{attribute 'GeneratedUsingTerminal: EK1100-0000-0018'}
{attribute addProperty BoxType "EK1100-0000-0018"}
{attribute addProperty Id "Beckhoff_EL72xxEK1122Beckhoff_EL72xxEK1122_A6E7F55E2A_0001_EL7201_0000_0017EL7201_91DE43F025A_0002_EL7201_0000_0018EL7201_91DE43F025A_0003_EL7201_0000_0019EL7201_91DE43F025A_0004_EL7201_0000_0020EL7201_91DE43F025A_0005_EL7201_0000_0021EL7201_91DE43F025A_0006_EL7201_0001_0017EL7201_24495B2825A_0007_EL7201_0001_0018EL7201_24495B2825A_0008_EL7201_0001_0019EL7201_24495B2825A_0009_EL7201_0001_0020EL7201_24495B2825A_0010_EL7201_0001_0021EL7201_24495B2825A_0011_EL7201_0010_0019EL7201_91DE43F025A_0012_EL7201_0010_0020EL7201_91DE43F025A_0013_EL7201_0010_0021EL7201_91DE43F025A_0014_EL7201_0010_0022EL7201_91DE43F025A_0015_EL7201_0010_0023EL7201_91DE43F025A_0016_EL7201_0010_0024EL7201_91DE43F025A_0017_EL7201_0010_0025EL7201_91DE43F025A_0018_EL7201_0010_0026EL7201_91DE43F025A_0019_EL7201_0010_0027EL7201_91DE43F025A_0020_EL7201_0010_0028EL7201_91DE43F025A_0021_EL7201_0010_0029EL7201_91DE43F025A_0022_EL7201_0010_0030EL7201_0985306B26A_0023_EL7201_0010_0031EL7201_0985306B26A_0024_EL7201_0010_0032EL7201_0985306B26A_0025_EL7201_0011_0019EL7201_24495B2825A_0026_EL7201_0011_0020EL7201_24495B2825A_0027_EL7201_0011_0021EL7201_24495B2825A_0028_EL7201_0011_0022EL7201_24495B2825A_0029_EL7201_0011_0023EL7201_24495B2825A_0030_EL7201_0011_0024EL7201_24495B2825A_0031_EL7201_0011_0025EL7201_24495B2825A_0032_EL7201_0011_0026EL7201_24495B2825A_0033_EL7201_0011_0027EL7201_24495B2825A_0034_EL7201_0011_0028EL7201_24495B2825A_0035_EL7201_0011_0029EL7201_24495B2825A_0036_EL7201_0011_0030EL7201_24495B2825A_0037_EL7201_0011_0031EL7201_24495B2825A_0038_EL7201_0011_0032EL7201_24495B2825A_0039_EL7211_0000_0020EL7211_91DE43F025A_0040_EL7211_0000_0021EL7211_91DE43F025A_0041_EL7211_0001_0020EL7211_24495B2825A_0042_EL7211_0001_0021EL7211_24495B2825A_0043_EL7211_0010_0023EL7211_91DE43F025A_0044_EL7211_0010_0024EL7211_91DE43F025A_0045_EL7211_0010_0025EL7211_91DE43F025A_0046_EL7211_0010_0026EL7211_91DE43F025A_0047_EL7211_0010_0027EL7211_91DE43F025A_0048_EL7211_0010_0028EL7211_91DE43F025A_0049_EL7211_0010_0029EL7211_91DE43F025A_0050_EL7211_0010_0030EL7211_0985306B26A_0051_EL7211_0010_0031EL7211_0985306B26A_0052_EL7211_0010_0032EL7211_0985306B26A_0053_EL7211_0011_0023EL7211_24495B2825A_0054_EL7211_0011_0024EL7211_24495B2825A_0055_EL7211_0011_0025EL7211_24495B2825A_0056_EL7211_0011_0026EL7211_24495B2825A_0057_EL7211_0011_0027EL7211_24495B2825A_0058_EL7211_0011_0028EL7211_24495B2825A_0059_EL7211_0011_0029EL7211_24495B2825A_0060_EL7211_0011_0030EL7211_24495B2825A_0061_EL7211_0011_0031EL7211_24495B2825A_0062_EL7211_0011_0032EL7211_24495B2825A_0063_EL7201_9014_0026EL7201_91DE43F025A_0064_EL7201_9014_0027EL7201_91DE43F025A_0065_EL7201_9014_0028EL7201_91DE43F025A_0066_EL7201_9014_0029EL7201_91DE43F025A_0067_EL7201_9014_0030EL7201_0985306B26A_0068_EL7201_9014_0031EL7201_0985306B26A_0069_EL7201_9014_0032EL7201_0985306B26A_0070_EL7201_9015_0026EL7201_24495B2825A_0071_EL7201_9015_0027EL7201_24495B2825A_0072_EL7201_9015_0028EL7201_24495B2825A_0073_EL7201_9015_0029EL7201_24495B2825A_0074_EL7201_9015_0030EL7201_24495B2825A_0075_EL7201_9015_0031EL7201_24495B2825A_0076_EL7201_9015_0032EL7201_24495B2825A_0077_EL7211_9014_0026EL7211_91DE43F025A_0078_EL7211_9014_0027EL7211_91DE43F025A_0079_EL7211_9014_0028EL7211_91DE43F025A_0080_EL7211_9014_0029EL7211_91DE43F025A_0081_EL7211_9014_0030EL7211_0985306B26A_0082_EL7211_9014_0031EL7211_0985306B26A_0083_EL7211_9014_0032EL7211_0985306B26A_0084_EL7211_9015_0026EL7211_24495B2825A_0085_EL7211_9015_0027EL7211_24495B2825A_0086_EL7211_9015_0028EL7211_24495B2825A_0087_EL7211_9015_0029EL7211_24495B2825A_0088_EL7211_9015_0030EL7211_24495B2825A_0089_EL7211_9015_0031EL7211_24495B2825A_0090_EL7211_9015_0032EL7211_24495B2825A_0091_EL7221_0000_0021EL7221_91DE43F025A_0092_EL7221_0001_0021EL7221_24495B2825A_0093_EL7221_9014_0028EL7221_91DE43F025A_0094_EL7221_9014_0029EL7221_91DE43F025A_0095_EL7221_9014_0030EL7221_0985306B26A_0096_EL7221_9014_0031EL7221_0985306B26A_0097_EL7221_9014_0032EL7221_0985306B26A_0098_EL7221_9015_0028EL7221_24495B2825A_0099_EL7221_9015_0029EL7221_24495B2825A_0100_EL7221_9015_0030EL7221_24495B2825A_0101_EL7221_9015_0031EL7221_24495B2825A_0102_EL7221_9015_0032EL7221_24495B2825"}
{attribute addProperty CRC "859834977"}
{attribute addProperty Size "2567"}
TYPE Beckhoff_EL72xx_33400A61 EXTENDS EK1100_1FC0878B :
STRUCT
	{attribute addProperty Name "Beckhoff_EL72xxEK1122"}
	{attribute addProperty PreviousPort "Beckhoff EL72xx : B"}
	Beckhoff_EL72xxEK1122 : Beckhoff_EL72xxEK1122_A6E7F55E;
	{attribute addProperty Name "A_0001_EL7201_0000_0017"}
	{attribute addProperty PreviousPort "Beckhoff EL72xxEK1122 : C"}
	A_0001_EL7201_0000_0017 : EL7201_91DE43F0;
	{attribute addProperty Name "A_0002_EL7201_0000_0018"}
	{attribute addProperty PreviousPort "A_0001(EL7201-0000-0017) : B"}
	A_0002_EL7201_0000_0018 : EL7201_91DE43F0;
	{attribute addProperty Name "A_0003_EL7201_0000_0019"}
	{attribute addProperty PreviousPort "A_0002(EL7201-0000-0018) : B"}
	A_0003_EL7201_0000_0019 : EL7201_91DE43F0;
	{attribute addProperty Name "A_0004_EL7201_0000_0020"}
	{attribute addProperty PreviousPort "A_0003(EL7201-0000-0019) : B"}
	A_0004_EL7201_0000_0020 : EL7201_91DE43F0;
	{attribute addProperty Name "A_0005_EL7201_0000_0021"}
	{attribute addProperty PreviousPort "A_0004(EL7201-0000-0020) : B"}
	A_0005_EL7201_0000_0021 : EL7201_91DE43F0;
	{attribute addProperty Name "A_0006_EL7201_0001_0017"}
	{attribute addProperty PreviousPort "A_0005(EL7201-0000-0021) : B"}
	A_0006_EL7201_0001_0017 : EL7201_24495B28;
	{attribute addProperty Name "A_0007_EL7201_0001_0018"}
	{attribute addProperty PreviousPort "A_0006(EL7201-0001-0017) : B"}
	A_0007_EL7201_0001_0018 : EL7201_24495B28;
	{attribute addProperty Name "A_0008_EL7201_0001_0019"}
	{attribute addProperty PreviousPort "A_0007(EL7201-0001-0018) : B"}
	A_0008_EL7201_0001_0019 : EL7201_24495B28;
	{attribute addProperty Name "A_0009_EL7201_0001_0020"}
	{attribute addProperty PreviousPort "A_0008(EL7201-0001-0019) : B"}
	A_0009_EL7201_0001_0020 : EL7201_24495B28;
	{attribute addProperty Name "A_0010_EL7201_0001_0021"}
	{attribute addProperty PreviousPort "A_0009(EL7201-0001-0020) : B"}
	A_0010_EL7201_0001_0021 : EL7201_24495B28;
	{attribute addProperty Name "A_0011_EL7201_0010_0019"}
	{attribute addProperty PreviousPort "A_0010(EL7201-0001-0021) : B"}
	A_0011_EL7201_0010_0019 : EL7201_91DE43F0;
	{attribute addProperty Name "A_0012_EL7201_0010_0020"}
	{attribute addProperty PreviousPort "A_0011(EL7201-0010-0019) : B"}
	A_0012_EL7201_0010_0020 : EL7201_91DE43F0;
	{attribute addProperty Name "A_0013_EL7201_0010_0021"}
	{attribute addProperty PreviousPort "A_0012(EL7201-0010-0020) : B"}
	A_0013_EL7201_0010_0021 : EL7201_91DE43F0;
	{attribute addProperty Name "A_0014_EL7201_0010_0022"}
	{attribute addProperty PreviousPort "A_0013(EL7201-0010-0021) : B"}
	A_0014_EL7201_0010_0022 : EL7201_91DE43F0;
	{attribute addProperty Name "A_0015_EL7201_0010_0023"}
	{attribute addProperty PreviousPort "A_0014(EL7201-0010-0022) : B"}
	A_0015_EL7201_0010_0023 : EL7201_91DE43F0;
	{attribute addProperty Name "A_0016_EL7201_0010_0024"}
	{attribute addProperty PreviousPort "A_0015(EL7201-0010-0023) : B"}
	A_0016_EL7201_0010_0024 : EL7201_91DE43F0;
	{attribute addProperty Name "A_0017_EL7201_0010_0025"}
	{attribute addProperty PreviousPort "A_0016(EL7201-0010-0024) : B"}
	A_0017_EL7201_0010_0025 : EL7201_91DE43F0;
	{attribute addProperty Name "A_0018_EL7201_0010_0026"}
	{attribute addProperty PreviousPort "A_0017(EL7201-0010-0025) : B"}
	A_0018_EL7201_0010_0026 : EL7201_91DE43F0;
	{attribute addProperty Name "A_0019_EL7201_0010_0027"}
	{attribute addProperty PreviousPort "A_0018(EL7201-0010-0026) : B"}
	A_0019_EL7201_0010_0027 : EL7201_91DE43F0;
	{attribute addProperty Name "A_0020_EL7201_0010_0028"}
	{attribute addProperty PreviousPort "A_0019(EL7201-0010-0027) : B"}
	A_0020_EL7201_0010_0028 : EL7201_91DE43F0;
	{attribute addProperty Name "A_0021_EL7201_0010_0029"}
	{attribute addProperty PreviousPort "A_0020(EL7201-0010-0028) : B"}
	A_0021_EL7201_0010_0029 : EL7201_91DE43F0;
	{attribute addProperty Name "A_0022_EL7201_0010_0030"}
	{attribute addProperty PreviousPort "A_0021(EL7201-0010-0029) : B"}
	A_0022_EL7201_0010_0030 : EL7201_0985306B;
	{attribute addProperty Name "A_0023_EL7201_0010_0031"}
	{attribute addProperty PreviousPort "A_0022(EL7201-0010-0030) : B"}
	A_0023_EL7201_0010_0031 : EL7201_0985306B;
	{attribute addProperty Name "A_0024_EL7201_0010_0032"}
	{attribute addProperty PreviousPort "A_0023(EL7201-0010-0031) : B"}
	A_0024_EL7201_0010_0032 : EL7201_0985306B;
	{attribute addProperty Name "A_0025_EL7201_0011_0019"}
	{attribute addProperty PreviousPort "A_0024(EL7201-0010-0032) : B"}
	A_0025_EL7201_0011_0019 : EL7201_24495B28;
	{attribute addProperty Name "A_0026_EL7201_0011_0020"}
	{attribute addProperty PreviousPort "A_0025(EL7201-0011-0019) : B"}
	A_0026_EL7201_0011_0020 : EL7201_24495B28;
	{attribute addProperty Name "A_0027_EL7201_0011_0021"}
	{attribute addProperty PreviousPort "A_0026(EL7201-0011-0020) : B"}
	A_0027_EL7201_0011_0021 : EL7201_24495B28;
	{attribute addProperty Name "A_0028_EL7201_0011_0022"}
	{attribute addProperty PreviousPort "A_0027(EL7201-0011-0021) : B"}
	A_0028_EL7201_0011_0022 : EL7201_24495B28;
	{attribute addProperty Name "A_0029_EL7201_0011_0023"}
	{attribute addProperty PreviousPort "A_0028(EL7201-0011-0022) : B"}
	A_0029_EL7201_0011_0023 : EL7201_24495B28;
	{attribute addProperty Name "A_0030_EL7201_0011_0024"}
	{attribute addProperty PreviousPort "A_0029(EL7201-0011-0023) : B"}
	A_0030_EL7201_0011_0024 : EL7201_24495B28;
	{attribute addProperty Name "A_0031_EL7201_0011_0025"}
	{attribute addProperty PreviousPort "A_0030(EL7201-0011-0024) : B"}
	A_0031_EL7201_0011_0025 : EL7201_24495B28;
	{attribute addProperty Name "A_0032_EL7201_0011_0026"}
	{attribute addProperty PreviousPort "A_0031(EL7201-0011-0025) : B"}
	A_0032_EL7201_0011_0026 : EL7201_24495B28;
	{attribute addProperty Name "A_0033_EL7201_0011_0027"}
	{attribute addProperty PreviousPort "A_0032(EL7201-0011-0026) : B"}
	A_0033_EL7201_0011_0027 : EL7201_24495B28;
	{attribute addProperty Name "A_0034_EL7201_0011_0028"}
	{attribute addProperty PreviousPort "A_0033(EL7201-0011-0027) : B"}
	A_0034_EL7201_0011_0028 : EL7201_24495B28;
	{attribute addProperty Name "A_0035_EL7201_0011_0029"}
	{attribute addProperty PreviousPort "A_0034(EL7201-0011-0028) : B"}
	A_0035_EL7201_0011_0029 : EL7201_24495B28;
	{attribute addProperty Name "A_0036_EL7201_0011_0030"}
	{attribute addProperty PreviousPort "A_0035(EL7201-0011-0029) : B"}
	A_0036_EL7201_0011_0030 : EL7201_24495B28;
	{attribute addProperty Name "A_0037_EL7201_0011_0031"}
	{attribute addProperty PreviousPort "A_0036(EL7201-0011-0030) : B"}
	A_0037_EL7201_0011_0031 : EL7201_24495B28;
	{attribute addProperty Name "A_0038_EL7201_0011_0032"}
	{attribute addProperty PreviousPort "A_0037(EL7201-0011-0031) : B"}
	A_0038_EL7201_0011_0032 : EL7201_24495B28;
	{attribute addProperty Name "A_0039_EL7211_0000_0020"}
	{attribute addProperty PreviousPort "A_0038(EL7201-0011-0032) : B"}
	A_0039_EL7211_0000_0020 : EL7211_91DE43F0;
	{attribute addProperty Name "A_0040_EL7211_0000_0021"}
	{attribute addProperty PreviousPort "A_0039(EL7211-0000-0020) : B"}
	A_0040_EL7211_0000_0021 : EL7211_91DE43F0;
	{attribute addProperty Name "A_0041_EL7211_0001_0020"}
	{attribute addProperty PreviousPort "A_0040(EL7211-0000-0021) : B"}
	A_0041_EL7211_0001_0020 : EL7211_24495B28;
	{attribute addProperty Name "A_0042_EL7211_0001_0021"}
	{attribute addProperty PreviousPort "A_0041(EL7211-0001-0020) : B"}
	A_0042_EL7211_0001_0021 : EL7211_24495B28;
	{attribute addProperty Name "A_0043_EL7211_0010_0023"}
	{attribute addProperty PreviousPort "A_0042(EL7211-0001-0021) : B"}
	A_0043_EL7211_0010_0023 : EL7211_91DE43F0;
	{attribute addProperty Name "A_0044_EL7211_0010_0024"}
	{attribute addProperty PreviousPort "A_0043(EL7211-0010-0023) : B"}
	A_0044_EL7211_0010_0024 : EL7211_91DE43F0;
	{attribute addProperty Name "A_0045_EL7211_0010_0025"}
	{attribute addProperty PreviousPort "A_0044(EL7211-0010-0024) : B"}
	A_0045_EL7211_0010_0025 : EL7211_91DE43F0;
	{attribute addProperty Name "A_0046_EL7211_0010_0026"}
	{attribute addProperty PreviousPort "A_0045(EL7211-0010-0025) : B"}
	A_0046_EL7211_0010_0026 : EL7211_91DE43F0;
	{attribute addProperty Name "A_0047_EL7211_0010_0027"}
	{attribute addProperty PreviousPort "A_0046(EL7211-0010-0026) : B"}
	A_0047_EL7211_0010_0027 : EL7211_91DE43F0;
	{attribute addProperty Name "A_0048_EL7211_0010_0028"}
	{attribute addProperty PreviousPort "A_0047(EL7211-0010-0027) : B"}
	A_0048_EL7211_0010_0028 : EL7211_91DE43F0;
	{attribute addProperty Name "A_0049_EL7211_0010_0029"}
	{attribute addProperty PreviousPort "A_0048(EL7211-0010-0028) : B"}
	A_0049_EL7211_0010_0029 : EL7211_91DE43F0;
	{attribute addProperty Name "A_0050_EL7211_0010_0030"}
	{attribute addProperty PreviousPort "A_0049(EL7211-0010-0029) : B"}
	A_0050_EL7211_0010_0030 : EL7211_0985306B;
	{attribute addProperty Name "A_0051_EL7211_0010_0031"}
	{attribute addProperty PreviousPort "A_0050(EL7211-0010-0030) : B"}
	A_0051_EL7211_0010_0031 : EL7211_0985306B;
	{attribute addProperty Name "A_0052_EL7211_0010_0032"}
	{attribute addProperty PreviousPort "A_0051(EL7211-0010-0031) : B"}
	A_0052_EL7211_0010_0032 : EL7211_0985306B;
	{attribute addProperty Name "A_0053_EL7211_0011_0023"}
	{attribute addProperty PreviousPort "A_0052(EL7211-0010-0032) : B"}
	A_0053_EL7211_0011_0023 : EL7211_24495B28;
	{attribute addProperty Name "A_0054_EL7211_0011_0024"}
	{attribute addProperty PreviousPort "A_0053(EL7211-0011-0023) : B"}
	A_0054_EL7211_0011_0024 : EL7211_24495B28;
	{attribute addProperty Name "A_0055_EL7211_0011_0025"}
	{attribute addProperty PreviousPort "A_0054(EL7211-0011-0024) : B"}
	A_0055_EL7211_0011_0025 : EL7211_24495B28;
	{attribute addProperty Name "A_0056_EL7211_0011_0026"}
	{attribute addProperty PreviousPort "A_0055(EL7211-0011-0025) : B"}
	A_0056_EL7211_0011_0026 : EL7211_24495B28;
	{attribute addProperty Name "A_0057_EL7211_0011_0027"}
	{attribute addProperty PreviousPort "A_0056(EL7211-0011-0026) : B"}
	A_0057_EL7211_0011_0027 : EL7211_24495B28;
	{attribute addProperty Name "A_0058_EL7211_0011_0028"}
	{attribute addProperty PreviousPort "A_0057(EL7211-0011-0027) : B"}
	A_0058_EL7211_0011_0028 : EL7211_24495B28;
	{attribute addProperty Name "A_0059_EL7211_0011_0029"}
	{attribute addProperty PreviousPort "A_0058(EL7211-0011-0028) : B"}
	A_0059_EL7211_0011_0029 : EL7211_24495B28;
	{attribute addProperty Name "A_0060_EL7211_0011_0030"}
	{attribute addProperty PreviousPort "A_0059(EL7211-0011-0029) : B"}
	A_0060_EL7211_0011_0030 : EL7211_24495B28;
	{attribute addProperty Name "A_0061_EL7211_0011_0031"}
	{attribute addProperty PreviousPort "A_0060(EL7211-0011-0030) : B"}
	A_0061_EL7211_0011_0031 : EL7211_24495B28;
	{attribute addProperty Name "A_0062_EL7211_0011_0032"}
	{attribute addProperty PreviousPort "A_0061(EL7211-0011-0031) : B"}
	A_0062_EL7211_0011_0032 : EL7211_24495B28;
	{attribute addProperty Name "A_0063_EL7201_9014_0026"}
	{attribute addProperty PreviousPort "A_0062(EL7211-0011-0032) : B"}
	A_0063_EL7201_9014_0026 : EL7201_91DE43F0;
	{attribute addProperty Name "A_0064_EL7201_9014_0027"}
	{attribute addProperty PreviousPort "A_0063(EL7201-9014-0026) : B"}
	A_0064_EL7201_9014_0027 : EL7201_91DE43F0;
	{attribute addProperty Name "A_0065_EL7201_9014_0028"}
	{attribute addProperty PreviousPort "A_0064(EL7201-9014-0027) : B"}
	A_0065_EL7201_9014_0028 : EL7201_91DE43F0;
	{attribute addProperty Name "A_0066_EL7201_9014_0029"}
	{attribute addProperty PreviousPort "A_0065(EL7201-9014-0028) : B"}
	A_0066_EL7201_9014_0029 : EL7201_91DE43F0;
	{attribute addProperty Name "A_0067_EL7201_9014_0030"}
	{attribute addProperty PreviousPort "A_0066(EL7201-9014-0029) : B"}
	A_0067_EL7201_9014_0030 : EL7201_0985306B;
	{attribute addProperty Name "A_0068_EL7201_9014_0031"}
	{attribute addProperty PreviousPort "A_0067(EL7201-9014-0030) : B"}
	A_0068_EL7201_9014_0031 : EL7201_0985306B;
	{attribute addProperty Name "A_0069_EL7201_9014_0032"}
	{attribute addProperty PreviousPort "A_0068(EL7201-9014-0031) : B"}
	A_0069_EL7201_9014_0032 : EL7201_0985306B;
	{attribute addProperty Name "A_0070_EL7201_9015_0026"}
	{attribute addProperty PreviousPort "A_0069(EL7201-9014-0032) : B"}
	A_0070_EL7201_9015_0026 : EL7201_24495B28;
	{attribute addProperty Name "A_0071_EL7201_9015_0027"}
	{attribute addProperty PreviousPort "A_0070(EL7201-9015-0026) : B"}
	A_0071_EL7201_9015_0027 : EL7201_24495B28;
	{attribute addProperty Name "A_0072_EL7201_9015_0028"}
	{attribute addProperty PreviousPort "A_0071(EL7201-9015-0027) : B"}
	A_0072_EL7201_9015_0028 : EL7201_24495B28;
	{attribute addProperty Name "A_0073_EL7201_9015_0029"}
	{attribute addProperty PreviousPort "A_0072(EL7201-9015-0028) : B"}
	A_0073_EL7201_9015_0029 : EL7201_24495B28;
	{attribute addProperty Name "A_0074_EL7201_9015_0030"}
	{attribute addProperty PreviousPort "A_0073(EL7201-9015-0029) : B"}
	A_0074_EL7201_9015_0030 : EL7201_24495B28;
	{attribute addProperty Name "A_0075_EL7201_9015_0031"}
	{attribute addProperty PreviousPort "A_0074(EL7201-9015-0030) : B"}
	A_0075_EL7201_9015_0031 : EL7201_24495B28;
	{attribute addProperty Name "A_0076_EL7201_9015_0032"}
	{attribute addProperty PreviousPort "A_0075(EL7201-9015-0031) : B"}
	A_0076_EL7201_9015_0032 : EL7201_24495B28;
	{attribute addProperty Name "A_0077_EL7211_9014_0026"}
	{attribute addProperty PreviousPort "A_0076(EL7201-9015-0032) : B"}
	A_0077_EL7211_9014_0026 : EL7211_91DE43F0;
	{attribute addProperty Name "A_0078_EL7211_9014_0027"}
	{attribute addProperty PreviousPort "A_0077(EL7211-9014-0026) : B"}
	A_0078_EL7211_9014_0027 : EL7211_91DE43F0;
	{attribute addProperty Name "A_0079_EL7211_9014_0028"}
	{attribute addProperty PreviousPort "A_0078(EL7211-9014-0027) : B"}
	A_0079_EL7211_9014_0028 : EL7211_91DE43F0;
	{attribute addProperty Name "A_0080_EL7211_9014_0029"}
	{attribute addProperty PreviousPort "A_0079(EL7211-9014-0028) : B"}
	A_0080_EL7211_9014_0029 : EL7211_91DE43F0;
	{attribute addProperty Name "A_0081_EL7211_9014_0030"}
	{attribute addProperty PreviousPort "A_0080(EL7211-9014-0029) : B"}
	A_0081_EL7211_9014_0030 : EL7211_0985306B;
	{attribute addProperty Name "A_0082_EL7211_9014_0031"}
	{attribute addProperty PreviousPort "A_0081(EL7211-9014-0030) : B"}
	A_0082_EL7211_9014_0031 : EL7211_0985306B;
	{attribute addProperty Name "A_0083_EL7211_9014_0032"}
	{attribute addProperty PreviousPort "A_0082(EL7211-9014-0031) : B"}
	A_0083_EL7211_9014_0032 : EL7211_0985306B;
	{attribute addProperty Name "A_0084_EL7211_9015_0026"}
	{attribute addProperty PreviousPort "A_0083(EL7211-9014-0032) : B"}
	A_0084_EL7211_9015_0026 : EL7211_24495B28;
	{attribute addProperty Name "A_0085_EL7211_9015_0027"}
	{attribute addProperty PreviousPort "A_0084(EL7211-9015-0026) : B"}
	A_0085_EL7211_9015_0027 : EL7211_24495B28;
	{attribute addProperty Name "A_0086_EL7211_9015_0028"}
	{attribute addProperty PreviousPort "A_0085(EL7211-9015-0027) : B"}
	A_0086_EL7211_9015_0028 : EL7211_24495B28;
	{attribute addProperty Name "A_0087_EL7211_9015_0029"}
	{attribute addProperty PreviousPort "A_0086(EL7211-9015-0028) : B"}
	A_0087_EL7211_9015_0029 : EL7211_24495B28;
	{attribute addProperty Name "A_0088_EL7211_9015_0030"}
	{attribute addProperty PreviousPort "A_0087(EL7211-9015-0029) : B"}
	A_0088_EL7211_9015_0030 : EL7211_24495B28;
	{attribute addProperty Name "A_0089_EL7211_9015_0031"}
	{attribute addProperty PreviousPort "A_0088(EL7211-9015-0030) : B"}
	A_0089_EL7211_9015_0031 : EL7211_24495B28;
	{attribute addProperty Name "A_0090_EL7211_9015_0032"}
	{attribute addProperty PreviousPort "A_0089(EL7211-9015-0031) : B"}
	A_0090_EL7211_9015_0032 : EL7211_24495B28;
	{attribute addProperty Name "A_0091_EL7221_0000_0021"}
	{attribute addProperty PreviousPort "A_0090(EL7211-9015-0032) : B"}
	A_0091_EL7221_0000_0021 : EL7221_91DE43F0;
	{attribute addProperty Name "A_0092_EL7221_0001_0021"}
	{attribute addProperty PreviousPort "A_0091(EL7221-0000-0021) : B"}
	A_0092_EL7221_0001_0021 : EL7221_24495B28;
	{attribute addProperty Name "A_0093_EL7221_9014_0028"}
	{attribute addProperty PreviousPort "A_0092(EL7221-0001-0021) : B"}
	A_0093_EL7221_9014_0028 : EL7221_91DE43F0;
	{attribute addProperty Name "A_0094_EL7221_9014_0029"}
	{attribute addProperty PreviousPort "A_0093(EL7221-9014-0028) : B"}
	A_0094_EL7221_9014_0029 : EL7221_91DE43F0;
	{attribute addProperty Name "A_0095_EL7221_9014_0030"}
	{attribute addProperty PreviousPort "A_0094(EL7221-9014-0029) : B"}
	A_0095_EL7221_9014_0030 : EL7221_0985306B;
	{attribute addProperty Name "A_0096_EL7221_9014_0031"}
	{attribute addProperty PreviousPort "A_0095(EL7221-9014-0030) : B"}
	A_0096_EL7221_9014_0031 : EL7221_0985306B;
	{attribute addProperty Name "A_0097_EL7221_9014_0032"}
	{attribute addProperty PreviousPort "A_0096(EL7221-9014-0031) : B"}
	A_0097_EL7221_9014_0032 : EL7221_0985306B;
	{attribute addProperty Name "A_0098_EL7221_9015_0028"}
	{attribute addProperty PreviousPort "A_0097(EL7221-9014-0032) : B"}
	A_0098_EL7221_9015_0028 : EL7221_24495B28;
	{attribute addProperty Name "A_0099_EL7221_9015_0029"}
	{attribute addProperty PreviousPort "A_0098(EL7221-9015-0028) : B"}
	A_0099_EL7221_9015_0029 : EL7221_24495B28;
	{attribute addProperty Name "A_0100_EL7221_9015_0030"}
	{attribute addProperty PreviousPort "A_0099(EL7221-9015-0029) : B"}
	A_0100_EL7221_9015_0030 : EL7221_24495B28;
	{attribute addProperty Name "A_0101_EL7221_9015_0031"}
	{attribute addProperty PreviousPort "A_0100(EL7221-9015-0030) : B"}
	A_0101_EL7221_9015_0031 : EL7221_24495B28;
	{attribute addProperty Name "A_0102_EL7221_9015_0032"}
	{attribute addProperty PreviousPort "A_0101(EL7221-9015-0031) : B"}
	A_0102_EL7221_9015_0032 : EL7221_24495B28;
END_STRUCT
END_TYPE

(* stored: Version 1.2.0.0, ProductVersion 3.1.4024.9
   DUT Beckhoff_EL72xx_33400A61: Id {ffd366c3-d41a-448a-919f-0e1df53cd5de} *)
